// TwinCAT 3 PLC project PLC_Project
// ProgramVersion: 3.1.4024.0
// libraries:
//   Lib, * (Terza-automation)
//   Tc2_Standard, * (Beckhoff Automation GmbH)
//   Tc2_System, * (Beckhoff Automation GmbH)
//   Tc2_Utilities, * (Beckhoff Automation GmbH)
//   Tc3_Module, * (Beckhoff Automation GmbH)
// project tree:
//   / PlcTask.TcTTO
//   POUs/ AI_OOR.TcPOU, AllCRAHs.TcPOU, AllEMeters.TcPOU, AlllDF.TcPOU, AllOtherDls.TcPOU, AllRTUStat.TcPOU, All_IO.TcPOU, MAIN.TcPOU, ModbusRTU.TcPOU, ScaleDP.TcPOU, SystemTime.TcPOU
// real-time tasks:
//   TASK PlcTask: cycle T#10ms, priority 20, ADS port 350
// I/O:
//   DEVICE Device 1 (EtherCAT)
// variable links:
//   PLC Project Instance <-> Device 1 (EtherCAT)/Term 1 (EK1100)
//     PlcTask Inputs/GVL_HW.CouplerStatus <-> InfoData/State
//   PLC Project Instance <-> Device 1 (EtherCAT)/Term 1 (EK1100)/Term 10 (EL1008)
//     PlcTask Inputs/GVL_HW.Term10Status <-> InfoData/State
//   PLC Project Instance <-> Device 1 (EtherCAT)/Term 1 (EK1100)/Term 11 (EL1008)
//     PlcTask Inputs/GVL_HW.Term11Status <-> InfoData/State
//   PLC Project Instance <-> Device 1 (EtherCAT)/Term 1 (EK1100)/Term 12 (EL1008)
//     PlcTask Inputs/GVL_HW.Term12Status <-> InfoData/State
//   PLC Project Instance <-> Device 1 (EtherCAT)/Term 1 (EK1100)/Term 13 (EL1008)
//     PlcTask Inputs/GVL_HW.Term13Status <-> InfoData/State
//   PLC Project Instance <-> Device 1 (EtherCAT)/Term 1 (EK1100)/Term 14 (EL1008)
//     PlcTask Inputs/GVL_HW.Term14Status <-> InfoData/State
//   PLC Project Instance <-> Device 1 (EtherCAT)/Term 1 (EK1100)/Term 15 (EL1008)
//     PlcTask Inputs/GVL_HW.Term15Status <-> InfoData/State
//   PLC Project Instance <-> Device 1 (EtherCAT)/Term 1 (EK1100)/Term 16 (EL1008)
//     PlcTask Inputs/GVL_HW.Term16Status <-> InfoData/State
//   PLC Project Instance <-> Device 1 (EtherCAT)/Term 1 (EK1100)/Term 17 (EL1008)
//     PlcTask Inputs/GVL_HW.Term17Status <-> InfoData/State
//   PLC Project Instance <-> Device 1 (EtherCAT)/Term 1 (EK1100)/Term 18 (EL1008)
//     PlcTask Inputs/GVL_HW.Term18Status <-> InfoData/State
//   PLC Project Instance <-> Device 1 (EtherCAT)/Term 1 (EK1100)/Term 19 (EL1008)
//     PlcTask Inputs/GVL_HW.Term19Status <-> InfoData/State
//   PLC Project Instance <-> Device 1 (EtherCAT)/Term 1 (EK1100)/Term 2 (EL1018)
//     PlcTask Inputs/GVL_HW.Term02Status <-> InfoData/State
//   PLC Project Instance <-> Device 1 (EtherCAT)/Term 1 (EK1100)/Term 20 (EL1008)
//     PlcTask Inputs/GVL_HW.Term20Status <-> InfoData/State
//   PLC Project Instance <-> Device 1 (EtherCAT)/Term 1 (EK1100)/Term 21 (EL1008)
//     PlcTask Inputs/GVL_HW.Term21Status <-> InfoData/State
//   PLC Project Instance <-> Device 1 (EtherCAT)/Term 1 (EK1100)/Term 22 (EL1008)
//     PlcTask Inputs/GVL_HW.Term22Status <-> InfoData/State
//   PLC Project Instance <-> Device 1 (EtherCAT)/Term 1 (EK1100)/Term 23 (EL9410)
//     PlcTask Inputs/GVL_HW.Term23Status <-> InfoData/State
//   PLC Project Instance <-> Device 1 (EtherCAT)/Term 1 (EK1100)/Term 24 (EL1008)
//     PlcTask Inputs/GVL_HW.Term24Status <-> InfoData/State
//   PLC Project Instance <-> Device 1 (EtherCAT)/Term 1 (EK1100)/Term 25 (EL1008)
//     PlcTask Inputs/GVL_HW.Term25Status <-> InfoData/State
//   PLC Project Instance <-> Device 1 (EtherCAT)/Term 1 (EK1100)/Term 26 (EL3058)
//     PlcTask Inputs/GVL_HW.Term26Status <-> InfoData/State
//   PLC Project Instance <-> Device 1 (EtherCAT)/Term 1 (EK1100)/Term 27 (EL6021)
//     PlcTask Inputs/GVL_HW.Term27Status <-> InfoData/State
//   PLC Project Instance <-> Device 1 (EtherCAT)/Term 1 (EK1100)/Term 28 (EL6021)
//     PlcTask Inputs/GVL_HW.Term28Status <-> InfoData/State
//   PLC Project Instance <-> Device 1 (EtherCAT)/Term 1 (EK1100)/Term 29 (EL6021)
//     PlcTask Inputs/GVL_HW.Term29Status <-> InfoData/State
//   PLC Project Instance <-> Device 1 (EtherCAT)/Term 1 (EK1100)/Term 3 (EL1008)
//     PlcTask Inputs/GVL_HW.Term03Status <-> InfoData/State
//   PLC Project Instance <-> Device 1 (EtherCAT)/Term 1 (EK1100)/Term 30 (EL6021)
//     PlcTask Inputs/GVL_HW.Term30Status <-> InfoData/State
//   PLC Project Instance <-> Device 1 (EtherCAT)/Term 1 (EK1100)/Term 31 (EL6021)
//     PlcTask Inputs/GVL_HW.Term31Status <-> COM TxPDO-Map Inputs/Status
//   PLC Project Instance <-> Device 1 (EtherCAT)/Term 1 (EK1100)/Term 32 (EL6021)
//     PlcTask Inputs/GVL_HW.Term32Status <-> COM TxPDO-Map Inputs/Status
//   PLC Project Instance <-> Device 1 (EtherCAT)/Term 1 (EK1100)/Term 33 (EL1018)
//     PlcTask Inputs/GVL_HW.Term33Status <-> InfoData/State
//   PLC Project Instance <-> Device 1 (EtherCAT)/Term 1 (EK1100)/Term 34 (EL1018)
//     PlcTask Inputs/GVL_HW.Term34Status <-> InfoData/State
//   PLC Project Instance <-> Device 1 (EtherCAT)/Term 1 (EK1100)/Term 4 (EL1008)
//     PlcTask Inputs/GVL_HW.Term04Status <-> InfoData/State
//   PLC Project Instance <-> Device 1 (EtherCAT)/Term 1 (EK1100)/Term 5 (EL1008)
//     PlcTask Inputs/GVL_HW.Term05Status <-> InfoData/State
//   PLC Project Instance <-> Device 1 (EtherCAT)/Term 1 (EK1100)/Term 6 (EL1008)
//     PlcTask Inputs/GVL_HW.Term06Status <-> InfoData/State
//   PLC Project Instance <-> Device 1 (EtherCAT)/Term 1 (EK1100)/Term 7 (EL1008)
//     PlcTask Inputs/GVL_HW.Term07Status <-> InfoData/State
//   PLC Project Instance <-> Device 1 (EtherCAT)/Term 1 (EK1100)/Term 8 (EL1008)
//     PlcTask Inputs/GVL_HW.Term08Status <-> InfoData/State
//   PLC Project Instance <-> Device 1 (EtherCAT)/Term 1 (EK1100)/Term 9 (EL1008)
//     PlcTask Inputs/GVL_HW.Term09Status <-> InfoData/State

CONFIGURATION PLC_Project
    RESOURCE PLC ON TwinCAT3
        TASK PlcTask(INTERVAL := T#10ms, PRIORITY := 20);
        PROGRAM MAIN WITH PlcTask : MAIN;
    END_RESOURCE
END_CONFIGURATION

// ---- POUs/MAIN.TcPOU
PROGRAM MAIN
VAR
	
	CRAHs : AllCRAHs;
	
	ModbusComms: ModbusRTU;
END_VAR

ModbusComms();

CRAHs();

END_PROGRAM

// ---- POUs/AllCRAHs.TcPOU
FUNCTION_BLOCK AllCRAHs
VAR
	OneCRAH : Lib.OneCRAH;
	CRAH_40_18_COM_ALM AT %I*: BOOL;
	CRAH_40_16_COM_ALM AT %I*: BOOL;
	CRAH_40_14_COM_ALM AT %I*: BOOL;
	CRAH_40_06_COM_ALM AT %I*: BOOL;
	CRAH_40_04_COM_ALM AT %I*: BOOL;
	CRAH_40_02_COM_ALM AT %I*: BOOL;
	CRAH_40_23_COM_ALM AT %I*: BOOL;
	CRAH_40_21_COM_ALM AT %I*: BOOL;
	CRAH_40_19_COM_ALM AT %I*: BOOL;
	CRAH_40_11_COM_ALM AT %I*: BOOL;
	CRAH_40_09_COM_ALM AT %I*: BOOL;
	CRAH_40_07_COM_ALM AT %I*: BOOL;
	CRAH_40_58_COM_ALM AT %I*: BOOL;
	CRAH_40_49_COM_ALM AT %I*: BOOL;
	CRAH_40_51_COM_ALM AT %I*: BOOL;
	CRAH_40_60_COM_ALM AT %I*: BOOL;
	
	
	CRAH_40_18_RUN_STS AT %I*: BOOL;
	CRAH_40_16_RUN_STS AT %I*: BOOL;
	CRAH_40_14_RUN_STS AT %I*: BOOL;
	CRAH_40_06_RUN_STS AT %I*: BOOL;
	CRAH_40_04_RUN_STS AT %I*: BOOL;
	CRAH_40_02_RUN_STS AT %I*: BOOL;
	CRAH_40_23_RUN_STS AT %I*: BOOL;
	CRAH_40_21_RUN_STS AT %I*: BOOL;
	CRAH_40_19_RUN_STS AT %I*: BOOL;
	CRAH_40_11_RUN_STS AT %I*: BOOL;
	CRAH_40_09_RUN_STS AT %I*: BOOL;
	CRAH_40_07_RUN_STS AT %I*: BOOL;
	CRAH_40_58_RUN_STS AT %I*: BOOL;
	CRAH_40_49_RUN_STS AT %I*: BOOL;
	CRAH_40_51_RUN_STS AT %I*: BOOL;
	CRAH_40_60_RUN_STS AT %I*: BOOL;
	
	
	CRAH_40_18_ISOL_1_STS AT %I*: BOOL;
	CRAH_40_18_ISOL_2_STS AT %I*: BOOL;	
	CRAH_40_16_ISOL_1_STS AT %I*: BOOL;
	CRAH_40_16_ISOL_2_STS AT %I*: BOOL;
	CRAH_40_14_ISOL_1_STS AT %I*: BOOL;
	CRAH_40_14_ISOL_2_STS AT %I*: BOOL;
	CRAH_40_06_ISOL_1_STS AT %I*: BOOL;
	CRAH_40_06_ISOL_2_STS AT %I*: BOOL;		
	CRAH_40_04_ISOL_1_STS AT %I*: BOOL;
	CRAH_40_04_ISOL_2_STS AT %I*: BOOL;	
	CRAH_40_02_ISOL_1_STS AT %I*: BOOL;
	CRAH_40_02_ISOL_2_STS AT %I*: BOOL;	
	CRAH_40_23_ISOL_1_STS AT %I*: BOOL;
	CRAH_40_23_ISOL_2_STS AT %I*: BOOL;	
	CRAH_40_21_ISOL_1_STS AT %I*: BOOL;
	CRAH_40_21_ISOL_2_STS AT %I*: BOOL;	
	CRAH_40_19_ISOL_1_STS AT %I*: BOOL;
	CRAH_40_19_ISOL_2_STS AT %I*: BOOL;
	CRAH_40_11_ISOL_1_STS AT %I*: BOOL;
	CRAH_40_11_ISOL_2_STS AT %I*: BOOL;
	CRAH_40_09_ISOL_1_STS AT %I*: BOOL;
	CRAH_40_09_ISOL_2_STS AT %I*: BOOL;	
	CRAH_40_07_ISOL_1_STS AT %I*: BOOL;
	CRAH_40_07_ISOL_2_STS AT %I*: BOOL;
	CRAH_40_58_ISOL_1_STS AT %I*: BOOL;
	CRAH_40_58_ISOL_2_STS AT %I*: BOOL;	
	CRAH_40_49_ISOL_1_STS AT %I*: BOOL;
	CRAH_40_49_ISOL_2_STS AT %I*: BOOL;	
	CRAH_40_51_ISOL_1_STS AT %I*: BOOL;
	CRAH_40_51_ISOL_2_STS AT %I*: BOOL;	
	CRAH_40_60_ISOL_1_STS AT %I*: BOOL;
	CRAH_40_60_ISOL_2_STS AT %I*: BOOL;
	
	CRAH_40_18: OneCRAH;
	CRAH_40_16: OneCRAH;
	CRAH_40_14: OneCRAH;
	CRAH_40_06: OneCRAH;
	
	CRAH_40_04: OneCRAH;
	CRAH_40_02: OneCRAH;
	CRAH_40_23: OneCRAH;
	CRAH_40_21: OneCRAH;
	
	CRAH_40_19: OneCRAH;
	CRAH_40_11: OneCRAH;
	CRAH_40_09: OneCRAH;
	CRAH_40_07: OneCRAH;
	
	CRAH_40_58: OneCRAH;
	CRAH_40_49: OneCRAH;
	CRAH_40_51: OneCRAH;
	CRAH_40_60: OneCRAH;
	
	AnyIOOffline: BOOL;

END_VAR


Lib.GVL.nInputCoilIndex      := Lib.GVL_DataHalls.StartInputCoilIndex_CRAH;
Lib.GVL.nOutputCoilIndex     := Lib.GVL_DataHalls.StartOutputCoilIndex_CRAH;
Lib.GVL.nInputRegisterIndex  := Lib.GVL_DataHalls.StartInputRegisterIndex_CRAH;
Lib.GVL.nOutputRegisterIndex := Lib.GVL_DataHalls.StartOutputRegisterIndex_CRAH;


AnyIOOffline:= Lib.GVl_hw.Term13Offline OR Lib.GVl_hw.Term15Offline OR Lib.GVl_hw.Term17Offline;
CRAH_40_18(
	Running:= CRAH_40_18_RUN_STS, 
	Alarm:= CRAH_40_18_COM_ALM, 
	Iso1_1_Sts:= CRAH_40_18_ISOL_1_STS, 
	Iso1_2_Sts:= CRAH_40_18_ISOL_2_STS, 
	Offline:= AnyIOOffline 
);

AnyIOOffline:= Lib.GVl_hw.Term13Offline OR Lib.GVl_hw.Term15Offline OR Lib.GVl_hw.Term17Offline;
CRAH_40_16(
	Running:= CRAH_40_16_RUN_STS, 
	Alarm:= CRAH_40_16_COM_ALM, 
	Iso1_1_Sts:= CRAH_40_16_ISOL_1_STS, 
	Iso1_2_Sts:= CRAH_40_16_ISOL_2_STS, 
	Offline:= AnyIOOffline 
);


AnyIOOffline:= Lib.GVl_hw.Term13Offline OR Lib.GVl_hw.Term15Offline OR Lib.GVl_hw.Term17Offline;
CRAH_40_14(
	Running:= CRAH_40_14_RUN_STS, 
	Alarm:= CRAH_40_14_COM_ALM, 
	Iso1_1_Sts:= CRAH_40_14_ISOL_1_STS, 
	Iso1_2_Sts:= CRAH_40_14_ISOL_2_STS, 
	Offline:= AnyIOOffline 
);


AnyIOOffline:= Lib.GVl_hw.Term13Offline OR Lib.GVl_hw.Term15Offline OR Lib.GVl_hw.Term18Offline;
CRAH_40_06(
	Running:= CRAH_40_06_RUN_STS, 
	Alarm:= CRAH_40_06_COM_ALM, 
	Iso1_1_Sts:= CRAH_40_06_ISOL_1_STS, 
	Iso1_2_Sts:= CRAH_40_06_ISOL_2_STS, 
	Offline:= AnyIOOffline 
);


AnyIOOffline:= Lib.GVl_hw.Term13Offline OR Lib.GVl_hw.Term15Offline OR Lib.GVl_hw.Term18Offline;
CRAH_40_04(
	Running:= CRAH_40_04_RUN_STS, 
	Alarm:= CRAH_40_04_COM_ALM, 
	Iso1_1_Sts:= CRAH_40_04_ISOL_1_STS, 
	Iso1_2_Sts:= CRAH_40_04_ISOL_2_STS, 
	Offline:= AnyIOOffline 
);


AnyIOOffline:= Lib.GVl_hw.Term13Offline OR Lib.GVl_hw.Term15Offline OR Lib.GVl_hw.Term18Offline;
CRAH_40_02(
	Running:= CRAH_40_02_RUN_STS, 
	Alarm:= CRAH_40_02_COM_ALM, 
	Iso1_1_Sts:= CRAH_40_02_ISOL_1_STS, 
	Iso1_2_Sts:= CRAH_40_02_ISOL_2_STS, 
	Offline:= AnyIOOffline 
);


AnyIOOffline:= Lib.GVl_hw.Term14Offline OR Lib.GVl_hw.Term16Offline OR Lib.GVl_hw.Term18Offline;
CRAH_40_23(
	Running:= CRAH_40_23_RUN_STS, 
	Alarm:= CRAH_40_23_COM_ALM, 
	Iso1_1_Sts:= CRAH_40_23_ISOL_1_STS, 
	Iso1_2_Sts:= CRAH_40_23_ISOL_2_STS, 
	Offline:= AnyIOOffline 
);


AnyIOOffline:= Lib.GVl_hw.Term14Offline OR Lib.GVl_hw.Term16Offline OR Lib.GVl_hw.Term19Offline;
CRAH_40_21(
	Running:= CRAH_40_21_RUN_STS, 
	Alarm:= CRAH_40_21_COM_ALM, 
	Iso1_1_Sts:= CRAH_40_21_ISOL_1_STS, 
	Iso1_2_Sts:= CRAH_40_21_ISOL_2_STS, 
	Offline:= AnyIOOffline 
);


AnyIOOffline:= Lib.GVl_hw.Term14Offline OR Lib.GVl_hw.Term16Offline OR Lib.GVl_hw.Term19Offline;
CRAH_40_19(
	Running:= CRAH_40_19_RUN_STS, 
	Alarm:= CRAH_40_19_COM_ALM, 
	Iso1_1_Sts:= CRAH_40_19_ISOL_1_STS, 
	Iso1_2_Sts:= CRAH_40_19_ISOL_2_STS, 
	Offline:= AnyIOOffline 
);


AnyIOOffline:= Lib.GVl_hw.Term14Offline OR Lib.GVl_hw.Term16Offline OR Lib.GVl_hw.Term19Offline;
CRAH_40_11(
	Running:= CRAH_40_11_RUN_STS, 
	Alarm:= CRAH_40_11_COM_ALM, 
	Iso1_1_Sts:= CRAH_40_11_ISOL_1_STS, 
	Iso1_2_Sts:= CRAH_40_11_ISOL_2_STS, 
	Offline:= AnyIOOffline 
);


AnyIOOffline:= Lib.GVl_hw.Term14Offline OR Lib.GVl_hw.Term16Offline OR Lib.GVl_hw.Term19Offline;
CRAH_40_09(
	Running:= CRAH_40_09_RUN_STS, 
	Alarm:= CRAH_40_09_COM_ALM, 
	Iso1_1_Sts:= CRAH_40_09_ISOL_1_STS, 
	Iso1_2_Sts:= CRAH_40_09_ISOL_2_STS, 
	Offline:= AnyIOOffline 
);


AnyIOOffline:= Lib.GVl_hw.Term14Offline OR Lib.GVl_hw.Term16Offline OR Lib.GVl_hw.Term19Offline;
CRAH_40_07(
	Running:= CRAH_40_07_RUN_STS, 
	Alarm:= CRAH_40_07_COM_ALM, 
	Iso1_1_Sts:= CRAH_40_07_ISOL_1_STS, 
	Iso1_2_Sts:= CRAH_40_07_ISOL_2_STS, 
	Offline:= AnyIOOffline 
);


AnyIOOffline:= Lib.GVl_hw.Term14Offline OR Lib.GVl_hw.Term16Offline OR Lib.GVl_hw.Term20Offline;
CRAH_40_58(
	Running:= CRAH_40_58_RUN_STS, 
	Alarm:= CRAH_40_58_COM_ALM, 
	Iso1_1_Sts:= CRAH_40_58_ISOL_1_STS, 
	Iso1_2_Sts:= FALSE, 
	Offline:= AnyIOOffline 
);


AnyIOOffline:= Lib.GVl_hw.Term14Offline OR Lib.GVl_hw.Term16Offline OR Lib.GVl_hw.Term20Offline;
CRAH_40_49(
	Running:= CRAH_40_49_RUN_STS, 
	Alarm:= CRAH_40_49_COM_ALM, 
	Iso1_1_Sts:= CRAH_40_49_ISOL_1_STS, 
	Iso1_2_Sts:= FALSE, 
	Offline:= AnyIOOffline 
);


AnyIOOffline:= Lib.GVl_hw.Term15Offline OR Lib.GVl_hw.Term17Offline OR Lib.GVl_hw.Term20Offline;
CRAH_40_51(
	Running:= CRAH_40_51_RUN_STS, 
	Alarm:= CRAH_40_51_COM_ALM, 
	Iso1_1_Sts:= CRAH_40_51_ISOL_1_STS, 
	Iso1_2_Sts:= FALSE, 
	Offline:= AnyIOOffline 
);


AnyIOOffline:= Lib.GVl_hw.Term15Offline OR Lib.GVl_hw.Term17Offline OR Lib.GVl_hw.Term20Offline;
CRAH_40_60(
	Running:= CRAH_40_60_RUN_STS, 
	Alarm:= CRAH_40_60_COM_ALM, 
	Iso1_1_Sts:= CRAH_40_60_ISOL_1_STS, 
	Iso1_2_Sts:= FALSE, 
	Offline:= AnyIOOffline 
);

END_FUNCTION_BLOCK

// ---- POUs/ModbusRTU.TcPOU
FUNCTION_BLOCK ModbusRTU
VAR
	MBComms1: ModbusRTU_THT;
	MBComms2: ModbusRTU_THT;
	MBComms3: ModbusRTU_THT;
	MBComms4: ModbusRTU_THT;
	MBComms5: ModbusRTU_EM_Integra;
END_VAR


MBComms1(MB_FirstUnitID:= 1, MB_LastUnitID:= 4);
MBComms2(MB_FirstUnitID:= 5, MB_LastUnitID:= 8);
MBComms3(MB_FirstUnitID:= 9, MB_LastUnitID:= 12);
MBComms4(MB_FirstUnitID:= 13, MB_LastUnitID:= 14);
MBComms5(MB_FirstUnitID:= 15, MB_LastUnitID:= 16);

END_FUNCTION_BLOCK

// ---- POUs/AI_OOR.TcPOU
FUNCTION AI_OOR : BOOL
VAR_INPUT
	Status : WORD;
END_VAR

// calculate whether the status for an analog input is indicating an error
// the error bit is the 7th bit of the status word
// access to bits is base 0, so the 7th bit is accessed with index 6

AI_OOR := Status.6;

END_FUNCTION

// ---- POUs/AllEMeters.TcPOU
FUNCTION_BLOCK AllEMeters
VAR
	OneEnergyMeter: Lib.OneEnergyMeter;
	
	EMeter_A: OneEnergyMeter;
	EMeter_B: OneEnergyMeter;
	


END_VAR


Lib.GVL.nInputCoilIndex:= Lib.GVL_DataHalls.StartInputCoilIndex_E_METER;
Lib.GVL.nOutputCoilIndex:= Lib.GVL_DataHalls.StartoutputCoilIndex_E_METER;
Lib.GVL.nInputRegisterIndex:= Lib.GVL_DataHalls.StartInputRegisterIndex_E_METER;
Lib.GVL.nOutputRegisterIndex:= Lib.GVL_DataHalls.StartOutputRegisterIndex_E_METER;


EMeter_A(
	Status:= Lib.GVL_EM.EM[1].Status, 
	Operating_Hrs:= Lib.GVL_EM.EM[1].Operating_Hrs, 
	Energy:= Lib.GVL_EM.EM[1].Energy, 
	Volume:= Lib.GVL_EM.EM[1].Volume, 
	Supply_Temp:= Lib.GVL_EM.EM[1].Supply_Temp, 
	Return_Temp:= Lib.GVL_EM.EM[1].Return_Temp, 
	Temp_Diff:= Lib.GVL_EM.EM[1].Temp_Diff, 
	Offline:= Lib.GVL_HW.Term31Offline OR Lib.GVL_EM.EM[1].CommsError);
	

EMeter_B(
	Status:= Lib.GVL_EM.EM[2].Status, 
	Operating_Hrs:= Lib.GVL_EM.EM[2].Operating_Hrs, 
	Energy:= Lib.GVL_EM.EM[2].Energy, 
	Volume:= Lib.GVL_EM.EM[2].Volume, 
	Supply_Temp:= Lib.GVL_EM.EM[2].Supply_Temp, 
	Return_Temp:= Lib.GVL_EM.EM[2].Return_Temp, 
	Temp_Diff:= Lib.GVL_EM.EM[2].Temp_Diff, 
	Offline:= Lib.GVL_HW.Term31Offline OR Lib.GVL_EM.EM[2].CommsError);

END_FUNCTION_BLOCK

// ---- POUs/AlllDF.TcPOU
FUNCTION_BLOCK AlllDF
VAR
	OneIDF: Lib.OneIDF;
	
	IDF17_3_A : OneIDF;
	
	IDF17_3_A_SPD_STS AT %I*: BOOL;
	IDF17_3_A_PF_ALM  AT %I*: BOOL;
	IDF17_3_A_115_BKR_STS AT %I*: BOOL;
	IDF17_3_A_115_BKR_TRIP_ALM AT %I*: BOOL;
	IDF17_3_A_125_BKR_STS AT %I*: BOOL;
	IDF17_3_A_125_BKR_TRIP_ALM AT %I*: BOOL;
	
	IDF14_3_B: OneIDF;
	
	IDF14_3_B_SPD_STS AT %I*: BOOL;
	IDF14_3_B_PF_ALM AT %I*: BOOL;
	IDF14_3_B_115_BKR_STS AT %I* : BOOL;
	IDF14_3_B_115_BKR_TRIP_ALM AT %I* : BOOL;
	IDF14_3_B_125_BKR_STS AT %I* : BOOL;
	IDF14_3_B_125_BKR_TRIP_ALM AT %I* : BOOL;
	
	IDF17_3_A_XT4S_10F1_TRIP_ALM AT %I* : BOOL;
	IDF14_3_B_XT4S_10F1_TRIP_ALM AT %I* : BOOL;
	
END_VAR

Lib.GVL.nInputCoilIndex:= Lib.GVL_DataHalls.StartInputCoilIndex_IDF;
Lib.GVL.nOutputCoilIndex:= Lib.GVL_DataHalls.StartOutputCoilIndex_IDF;
Lib.GVL.nInputRegisterIndex:= Lib.GVL_DataHalls.StartInputRegisterIndex_IDF;
Lib.GVL.nOutputRegisterIndex:= Lib.GVL_DataHalls.StartOutputRegisterIndex_IDF;


IDF17_3_A(
	sur_STS:= IDF17_3_A_SPD_STS, 
	phs_ALM:= IDF17_3_A_PF_ALM, 
	sur_phs_offline:= Lib.GVL_HW.Term20Offline, 
	BRK115_POS_STS:= IDF17_3_A_115_BKR_STS, 
	BRK115_TRIP_ALM:= IDF17_3_A_115_BKR_TRIP_ALM, 
	BRK115_offline:= Lib.GVL_HW.Term20Offline, 
	BRK125_POS_STS:= IDF17_3_A_125_BKR_STS, 
	BRK125_TRIP_ALM:= IDF17_3_A_125_BKR_TRIP_ALM, 
	BRK125_offline:= Lib.GVL_HW.Term20Offline, 
	INCOMER_TRIP_ALM:= IDF17_3_A_XT4S_10F1_TRIP_ALM, 
	INCOMER_offline:= Lib.GVL_HW.Term21Offline);
	
	
IDF14_3_B(
	sur_STS:= IDF14_3_B_SPD_STS, 
	phs_ALM:= IDF14_3_B_PF_ALM, 
	sur_phs_offline:= Lib.GVL_HW.Term20Offline, 
	BRK115_POS_STS:= IDF14_3_B_115_BKR_STS, 
	BRK115_TRIP_ALM:= IDF14_3_B_115_BKR_TRIP_ALM, 
	BRK115_offline:= Lib.GVL_HW.Term30Offline, 
	BRK125_POS_STS:= IDF14_3_B_125_BKR_STS, 
	BRK125_TRIP_ALM:= IDF14_3_B_125_BKR_TRIP_ALM, 
	BRK125_offline:= Lib.GVL_HW.Term30Offline, 
	INCOMER_TRIP_ALM:= IDF14_3_B_XT4S_10F1_TRIP_ALM, 
	INCOMER_offline:= Lib.GVL_HW.Term21Offline);

END_FUNCTION_BLOCK

// ---- POUs/AllOtherDls.TcPOU
FUNCTION_BLOCK AllOtherDls
VAR
	OneDI: Lib.OneDI;
	
	PSU1_ALM AT %I* : BOOL;
	PSU2_ALM AT %I* : BOOL;
	FAP_PNL_ALM AT %I* : BOOL;
	FAP_LOOP_ALM AT %I* : BOOL;
	Telco_ASD_A_PNL_ALM AT %I* : BOOL;
	Telco_ASD_B_PNL_ALM AT %I* : BOOL;
	DH_ASD_PNL_ALM AT %I* : BOOL;

	
	PSU1_Healthy: OneDI;
	PSU2_Healthy: OneDI;
	FAP_Healthy: OneDI;
	FAPL_Healthy: OneDI;
	TelcoSDP_A_Healthy: OneDI;
	TelcoSDP_B_Healthy: OneDI;
	DHSDP_Healthy: OneDI;
	
	UPS_BAT_LOW_ALM AT %I* : BOOL;
	UPS_BAT_MODE AT %I* : BOOL;
	
	UPS_BatLow: OneDI;
	UPS_BatMode: OneDI;

END_VAR

PSU1_Healthy(Value:= PSU1_ALM, Offline:= Lib.GVL_HW.Term13Offline);

PSU2_Healthy(Value:= PSU2_ALM , Offline:= Lib.GVL_HW.Term13Offline);

FAP_Healthy (Value:= FAP_PNL_ALM , Offline:= Lib.GVL_HW.Term20Offline);

FAPL_Healthy(Value:= FAP_LOOP_ALM, Offline:= Lib.GVL_HW.Term20Offline);

TelcoSDP_A_Healthy(Value:= Telco_ASD_A_PNL_ALM, Offline:= Lib.GVL_HW.Term21Offline);

TelcoSDP_B_Healthy(Value:= TelcoSDP_B_Healthy , Offline:= Lib.GVL_HW.Term21Offline);

DHSDP_Healthy(Value:= DH_ASD_PNL_ALM , Offline:= Lib.GVL_HW.Term21Offline);

UPS_BatLow(Value:= UPS_BAT_LOW_ALM, Offline:= Lib.GVL_HW.Term21Offline );

UPS_BatMode(Value:= UPS_BAT_MODE , Offline:= Lib.GVL_HW.Term21Offline);

END_FUNCTION_BLOCK

// ---- POUs/AllRTUStat.TcPOU
FUNCTION_BLOCK AllRTUStat
VAR
	i:INT;
END_VAR

Lib.GVL.nInputCoilIndex:= Lib.GVL_DataHalls.StartInputCoilIndex_RTUStat;
Lib.GVL.nOutputCoilIndex:= Lib.GVL_DataHalls.StartOutputCoilIndex_RTUStat;
Lib.GVL.nInputRegisterIndex:= Lib.GVL_DataHalls.StartInputRegisterIndex_RTUStat;
Lib.GVL.nOutputRegisterIndex:= Lib.GVL_DataHalls.StartOutputRegisterIndex_RTUStat;

i := Lib.GVL.nInputCoilIndex;

Lib.GVL.mb_Input_Coils[i+0] := Lib.GVL_THT.THT[1].CommsError;
Lib.GVL.mb_Input_Coils[i+1] := Lib.GVL_THT.THT[2].CommsError;
Lib.GVL.mb_Input_Coils[i+2] := Lib.GVL_THT.THT[3].CommsError;
Lib.GVL.mb_Input_Coils[i+3] := Lib.GVL_THT.THT[4].CommsError;
Lib.GVL.mb_Input_Coils[i+4] := Lib.GVL_THT.THT[5].CommsError;
Lib.GVL.mb_Input_Coils[i+5] := Lib.GVL_THT.THT[6].CommsError;
Lib.GVL.mb_Input_Coils[i+6] := Lib.GVL_THT.THT[7].CommsError;
Lib.GVL.mb_Input_Coils[i+7] := Lib.GVL_THT.THT[8].CommsError;
Lib.GVL.mb_Input_Coils[i+8] := Lib.GVL_THT.THT[9].CommsError;
Lib.GVL.mb_Input_Coils[i+9] := Lib.GVL_THT.THT[10].CommsError;
Lib.GVL.mb_Input_Coils[i+10]:= Lib.GVL_THT.THT[11].CommsError;
Lib.GVL.mb_Input_Coils[i+11]:= Lib.GVL_THT.THT[12].CommsError;
Lib.GVL.mb_Input_Coils[i+12]:= Lib.GVL_THT.THT[13].CommsError;
Lib.GVL.mb_Input_Coils[i+13]:= Lib.GVL_THT.THT[14].CommsError;

Lib.GVL.mb_Input_Coils[i+14]:= Lib.GVL_EM.EM[1].CommsError;
Lib.GVL.mb_Input_Coils[i+15]:= Lib.GVL_EM.EM[2].CommsError;

Lib.GVL.mb_Input_Registers[i+0] := INT_TO_WORD(Lib.GVL_THT.THT[1].CommsErrorCode);
Lib.GVL.mb_Input_Registers[i+1] := INT_TO_WORD(Lib.GVL_THT.THT[2].CommsErrorCode);
Lib.GVL.mb_Input_Registers[i+2] := INT_TO_WORD(Lib.GVL_THT.THT[3].CommsErrorCode);
Lib.GVL.mb_Input_Registers[i+3] := INT_TO_WORD(Lib.GVL_THT.THT[4].CommsErrorCode);
Lib.GVL.mb_Input_Registers[i+4] := INT_TO_WORD(Lib.GVL_THT.THT[5].CommsErrorCode);
Lib.GVL.mb_Input_Registers[i+5] := INT_TO_WORD(Lib.GVL_THT.THT[6].CommsErrorCode);
Lib.GVL.mb_Input_Registers[i+6] := INT_TO_WORD(Lib.GVL_THT.THT[7].CommsErrorCode);
Lib.GVL.mb_Input_Registers[i+7] := INT_TO_WORD(Lib.GVL_THT.THT[8].CommsErrorCode);
Lib.GVL.mb_Input_Registers[i+8] := INT_TO_WORD(Lib.GVL_THT.THT[9].CommsErrorCode);
Lib.GVL.mb_Input_Registers[i+9] := INT_TO_WORD(Lib.GVL_THT.THT[10].CommsErrorCode);
Lib.GVL.mb_Input_Registers[i+10]:= INT_TO_WORD(Lib.GVL_THT.THT[11].CommsErrorCode);
Lib.GVL.mb_Input_Registers[i+11]:= INT_TO_WORD(Lib.GVL_THT.THT[12].CommsErrorCode);
Lib.GVL.mb_Input_Registers[i+12]:= INT_TO_WORD(Lib.GVL_THT.THT[13].CommsErrorCode);
Lib.GVL.mb_Input_Registers[i+13]:= INT_TO_WORD(Lib.GVL_THT.THT[14].CommsErrorCode);

Lib.GVL.mb_Input_Registers[i+14]:= INT_TO_WORD(Lib.GVL_THT.THT[15].CommsErrorCode);
Lib.GVL.mb_Input_Registers[i+15]:= INT_TO_WORD(Lib.GVL_THT.THT[16].CommsErrorCode);

END_FUNCTION_BLOCK

// ---- POUs/All_IO.TcPOU
FUNCTION_BLOCK All_IO
VAR_TEMP
	i : INT;
END_VAR

Lib.GVL_HW.CouplerOffline:= NOT Lib.GVL_HW.CouplerStatus.3;
Lib.GVL_HW.Term02Offline := NOT Lib.GVL_HW.Term02Status.3;
Lib.GVL_HW.Term03Offline := NOT Lib.GVL_HW.Term03Status.3;
Lib.GVL_HW.Term04Offline := NOT Lib.GVL_HW.Term04Status.3;
Lib.GVL_HW.Term05Offline := NOT Lib.GVL_HW.Term05Status.3;
Lib.GVL_HW.Term06Offline := NOT Lib.GVL_HW.Term06Status.3;
Lib.GVL_HW.Term07Offline := NOT Lib.GVL_HW.Term07Status.3;
Lib.GVL_HW.Term08Offline := NOT Lib.GVL_HW.Term08Status.3;
Lib.GVL_HW.Term09Offline := NOT Lib.GVL_HW.Term09Status.3;
Lib.GVL_HW.Term10Offline := NOT Lib.GVL_HW.Term10Status.3;
Lib.GVL_HW.Term11Offline := NOT Lib.GVL_HW.Term11Status.3;
Lib.GVL_HW.Term12Offline := NOT Lib.GVL_HW.Term12Status.3;
Lib.GVL_HW.Term13Offline := NOT Lib.GVL_HW.Term13Status.3;
Lib.GVL_HW.Term14Offline := NOT Lib.GVL_HW.Term14Status.3;
Lib.GVL_HW.Term15Offline := NOT Lib.GVL_HW.Term15Status.3;
Lib.GVL_HW.Term16Offline := NOT Lib.GVL_HW.Term16Status.3;
Lib.GVL_HW.Term17Offline := NOT Lib.GVL_HW.Term17Status.3;
Lib.GVL_HW.Term18Offline := NOT Lib.GVL_HW.Term18Status.3;
Lib.GVL_HW.Term19Offline := NOT Lib.GVL_HW.Term19Status.3;
Lib.GVL_HW.Term20Offline := NOT Lib.GVL_HW.Term20Status.3;
Lib.GVL_HW.Term21Offline := NOT Lib.GVL_HW.Term21Status.3;
Lib.GVL_HW.Term22Offline := NOT Lib.GVL_HW.Term22Status.3;
Lib.GVL_HW.Term23Offline := NOT Lib.GVL_HW.Term23Status.3;
Lib.GVL_HW.Term24Offline := NOT Lib.GVL_HW.Term24Status.3;
Lib.GVL_HW.Term25Offline := NOT Lib.GVL_HW.Term25Status.3;
Lib.GVL_HW.Term26Offline := NOT Lib.GVL_HW.Term26Status.3;
Lib.GVL_HW.Term27Offline := NOT Lib.GVL_HW.Term27Status.3;
Lib.GVL_HW.Term28Offline := NOT Lib.GVL_HW.Term28Status.3;
Lib.GVL_HW.Term29Offline := NOT Lib.GVL_HW.Term29Status.3;
Lib.GVL_HW.Term30Offline := NOT Lib.GVL_HW.Term30Status.3;
Lib.GVL_HW.Term31Offline := NOT Lib.GVL_HW.Term31Status.3;
Lib.GVL_HW.Term32Offline := NOT Lib.GVL_HW.Term32Status.3;
Lib.GVL_HW.Term33Offline := NOT Lib.GVL_HW.Term33Status.3;
Lib.GVL_HW.Term34Offline := NOT Lib.GVL_HW.Term34Status.3;

Lib.GVL.nInputCoilIndex := lib.GVL_DataHalls.StartInputCoilIndex_IO;
Lib.GVL.nOutputCoilIndex:= lib.GVL_DataHalls.StartOutputCoilIndex_IO;
Lib.GVL.nInputRegisterIndex := lib.GVL_DataHalls.StartInputCoilIndex_IO;
Lib.GVL.nOutputRegisterIndex:= lib.GVL_DataHalls.StartOutputCoilIndex_IO;


i:= lib.GVL.nInputCoilIndex;

Lib.GVL.mb_Input_Coils[i+0] := Lib.GVL_HW.CouplerOffline;
Lib.GVL.mb_Input_Coils[i+1] := Lib.GVL_HW.Term02Offline;
Lib.GVL.mb_Input_Coils[i+2] := Lib.GVL_HW.Term03Offline;
Lib.GVL.mb_Input_Coils[i+3] := Lib.GVL_HW.Term04Offline;
Lib.GVL.mb_Input_Coils[i+4] := Lib.GVL_HW.Term05Offline;
Lib.GVL.mb_Input_Coils[i+5] := Lib.GVL_HW.Term06Offline;
Lib.GVL.mb_Input_Coils[i+6] := Lib.GVL_HW.Term07Offline;
Lib.GVL.mb_Input_Coils[i+7] := Lib.GVL_HW.Term08Offline;
Lib.GVL.mb_Input_Coils[i+8] := Lib.GVL_HW.Term09Offline;
Lib.GVL.mb_Input_Coils[i+9] := Lib.GVL_HW.Term10Offline;
Lib.GVL.mb_Input_Coils[i+10]:= Lib.GVL_HW.Term11Offline;
Lib.GVL.mb_Input_Coils[i+11]:= Lib.GVL_HW.Term12Offline;
Lib.GVL.mb_Input_Coils[i+12]:= Lib.GVL_HW.Term13Offline;
Lib.GVL.mb_Input_Coils[i+13]:= Lib.GVL_HW.Term14Offline;
Lib.GVL.mb_Input_Coils[i+14]:= Lib.GVL_HW.Term15Offline;
Lib.GVL.mb_Input_Coils[i+15]:= Lib.GVL_HW.Term16Offline;
Lib.GVL.mb_Input_Coils[i+16]:= Lib.GVL_HW.Term17Offline;
Lib.GVL.mb_Input_Coils[i+17]:= Lib.GVL_HW.Term18Offline;
Lib.GVL.mb_Input_Coils[i+18]:= Lib.GVL_HW.Term19Offline;
Lib.GVL.mb_Input_Coils[i+19]:= Lib.GVL_HW.Term20Offline;
Lib.GVL.mb_Input_Coils[i+20]:= Lib.GVL_HW.Term21Offline;
Lib.GVL.mb_Input_Coils[i+21]:= Lib.GVL_HW.Term22Offline;
Lib.GVL.mb_Input_Coils[i+22]:= Lib.GVL_HW.Term23Offline;
Lib.GVL.mb_Input_Coils[i+23]:= Lib.GVL_HW.Term24Offline;
Lib.GVL.mb_Input_Coils[i+24]:= Lib.GVL_HW.Term25Offline;
Lib.GVL.mb_Input_Coils[i+25]:= Lib.GVL_HW.Term26Offline;
Lib.GVL.mb_Input_Coils[i+26]:= Lib.GVL_HW.Term27Offline;
Lib.GVL.mb_Input_Coils[i+27]:= Lib.GVL_HW.Term28Offline;
Lib.GVL.mb_Input_Coils[i+28]:= Lib.GVL_HW.Term29Offline;
Lib.GVL.mb_Input_Coils[i+29]:= Lib.GVL_HW.Term30Offline;
Lib.GVL.mb_Input_Coils[i+30]:= Lib.GVL_HW.Term31Offline;
Lib.GVL.mb_Input_Coils[i+31]:= Lib.GVL_HW.Term32Offline;
Lib.GVL.mb_Input_Coils[i+32]:= Lib.GVL_HW.Term33Offline;
Lib.GVL.mb_Input_Coils[i+33]:= Lib.GVL_HW.Term34Offline;
Lib.GVL.mb_Input_Coils[i+34]:= TRUE;
Lib.GVL.mb_Input_Coils[i+35]:= TRUE;
Lib.GVL.mb_Input_Coils[i+36]:= TRUE;
Lib.GVL.mb_Input_Coils[i+37]:= TRUE;
Lib.GVL.mb_Input_Coils[i+38]:= TRUE;
Lib.GVL.mb_Input_Coils[i+39]:= TRUE;

END_FUNCTION_BLOCK

// ---- POUs/ScaleDP.TcPOU
FUNCTION ScaleDP : real
VAR_INPUT
	AIValue: WORD;
END_VAR


// Raw value of 0 to 32767 scales to -50 to +50
ScaleDP:= WORD_TO_REAL(AIValue) / 327.67 - 50.0;

END_FUNCTION

// ---- POUs/SystemTime.TcPOU
FUNCTION_BLOCK SystemTime
VAR_INPUT
END_VAR
VAR_OUTPUT
END_VAR
VAR
END_VAR


Lib.GVL_HW.fbGetLocalSystemTime(
	sNetID:= , 
	bEnable:= TRUE, 
	dwCycle:= 1, 
	dwOpt:= , 
	tTimeout:= , 
	bValid=> , 
	systemTime=> , 
	tzID=> );
	
Lib.GVL_HW.sSystemTime:= SYSTEMTIME_TO_STRING(Lib.GVL_HW.fbGetLocalSystemTime.systemTime);
Lib.GVL_HW.sSystemDate:=MID(STR:= Lib.GVL_HW.sSystemTime, LEN:= 10, POS:= 1);
Lib.GVL_HW.sSystemDate:=MID(STR:= Lib.GVL_HW.sSystemTime, LEN:= 8, POS:= 12);

END_FUNCTION_BLOCK
